(* Logix 5000 project; controller Sucrose_Main Emulate 5570 rev 20.12; software revision 20.01; part 7 of 30 *)
(* tags used below, declared in another part *)
   Alarm_ACK_Master_Timer : TIMER;
   DI_E23_5 : ALIAS FOR FLX_E23:5:I;   // Discrete Input EN2T_FLX 192.168.1.23
   DI_E25_3 : ALIAS FOR FLX_E25:3:I;   // Discrete Input EN2T_FLX 192.168.1.25
   DO_E24_2 : ALIAS FOR FLX_E24:2:O;   // Discrete Output EN2T_FLX 192.168.1.24
   DO_E25_4 : ALIAS FOR FLX_E25:4:O;   // Discrete Output EN2T_FLX 192.168.1.25
   DO_E25_5 : ALIAS FOR FLX_E25:5:O;   // Discrete Output EN2T_FLX 192.168.1.25
   FV610010_AOI : QSI_Flow_Valve;   // CIP SUPPLY TO RECEIVING PUMP #1
   FV610020_AOI : QSI_Flow_Valve;   // CIP SUPPLY TO RECEIVING PUMP #2
   FV610030_AOI : QSI_Flow_Valve;   // LOW POINT DRAIN VALVE
   FV610401_AOI : QSI_Flow_Valve;   // FV-61-04-01-O VALVE MANIFOLD TO SUCROSE TRANSFER PUMP #1 VALVE OPEN
   FV610402_AOI : QSI_Flow_Valve;   // FV-61-04-02-O VALVE MANIFOLD TO SUCROSE TRANSFER PUMP #2 VALVE OPEN
   FV620010_AOI : QSI_Flow_Valve;   // FV-62-00-10-O RECEIVING PUMP #1 TO CIP RETURN MIX PROOF VALVE OPEN
   FV620020_AOI : QSI_Flow_Valve;   // FV-62-00-20-O RECEIVING PUMP #2 TO CIP RETURN MIX PROOF VALVE OPEN
   FV620701_AOI : QSI_Flow_Valve;   // FV-62-07-01-O SUCROSE RING MAIN RETURN TO CIP RETURN VALVE VALVE OPEN
   FV621001_AOI : QSI_Flow_Valve;   // FV-62-10-01-O SUCROSE RECEIVING TO CIP RETURN VALVE OPEN
   Sucrose_MM_Enable : BOOL;
   SucroseCIP_P230401_REMOTE : CIP_REMOTE;
   SucroseCIP_P230402_REMOTE : CIP_REMOTE;
   SucroseCIP_RECEIVING2_REMOTE : CIP_REMOTE;
   SucroseCIP_RECEIVING_LINE_REMOTE : CIP_REMOTE;
   SucroseCIP_RECEIVING_REMOTE : CIP_REMOTE;
   SucroseCIP_RINGMAIN_REMOTE : CIP_REMOTE;
(* CIP_RemoteArea_EN2T_IO_Discrete_DO_E24_1, continued *)

ROUTINE MainRoutine   (* ladder *)
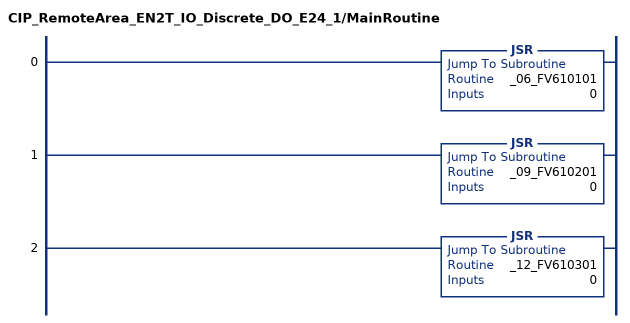
   0: JSR(_06_FV610101,0);
   1: JSR(_09_FV610201,0);
   2: JSR(_12_FV610301,0);
END_ROUTINE
END_PROGRAM

PROGRAM CIP_RemoteArea_EN2T_IO_Discrete_DO_E24_2   (* main routine MainRoutine *)

ROUTINE _00_FV610401   (* ladder *)
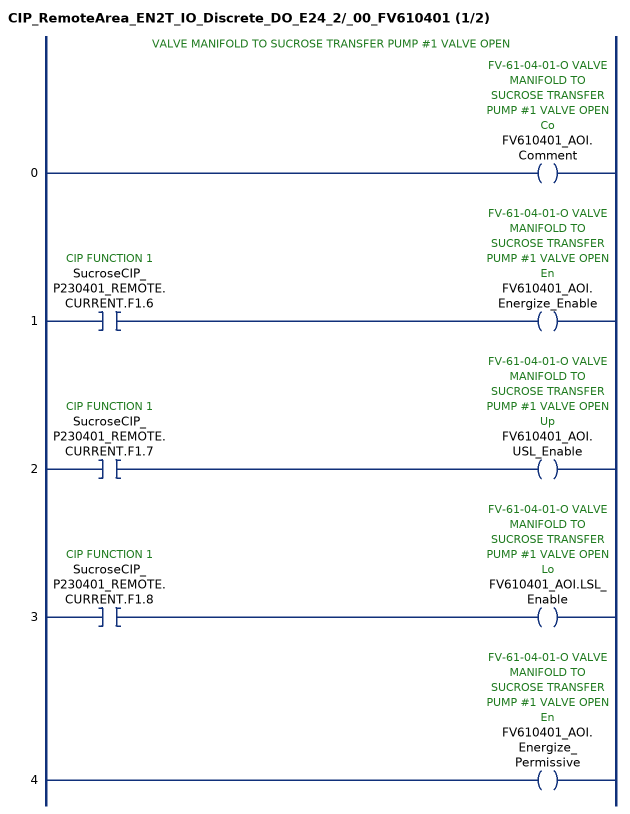
   // VALVE MANIFOLD TO SUCROSE TRANSFER PUMP #1 VALVE OPEN
   0: OTE(FV610401_AOI.Comment);
   1: XIC(SucroseCIP_P230401_REMOTE.CURRENT.F1.6)OTE(FV610401_AOI.Energize_Enable);
   2: XIC(SucroseCIP_P230401_REMOTE.CURRENT.F1.7)OTE(FV610401_AOI.USL_Enable);
   3: XIC(SucroseCIP_P230401_REMOTE.CURRENT.F1.8)OTE(FV610401_AOI.LSL_Enable);
   4: OTE(FV610401_AOI.Energize_Permissive);
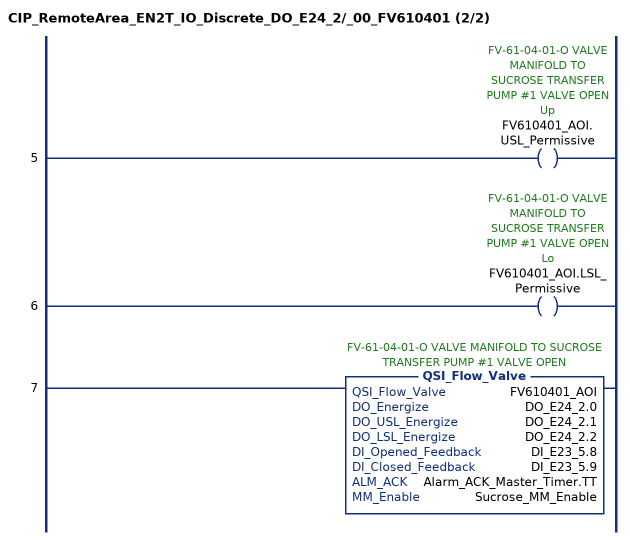
   5: OTE(FV610401_AOI.USL_Permissive);
   6: OTE(FV610401_AOI.LSL_Permissive);
   7: QSI_Flow_Valve(FV610401_AOI,DO_E24_2.0,DO_E24_2.1,DO_E24_2.2,DI_E23_5.8,DI_E23_5.9,Alarm_ACK_Master_Timer.TT,Sucrose_MM_Enable);
END_ROUTINE

ROUTINE _03_FV610402   (* ladder *)
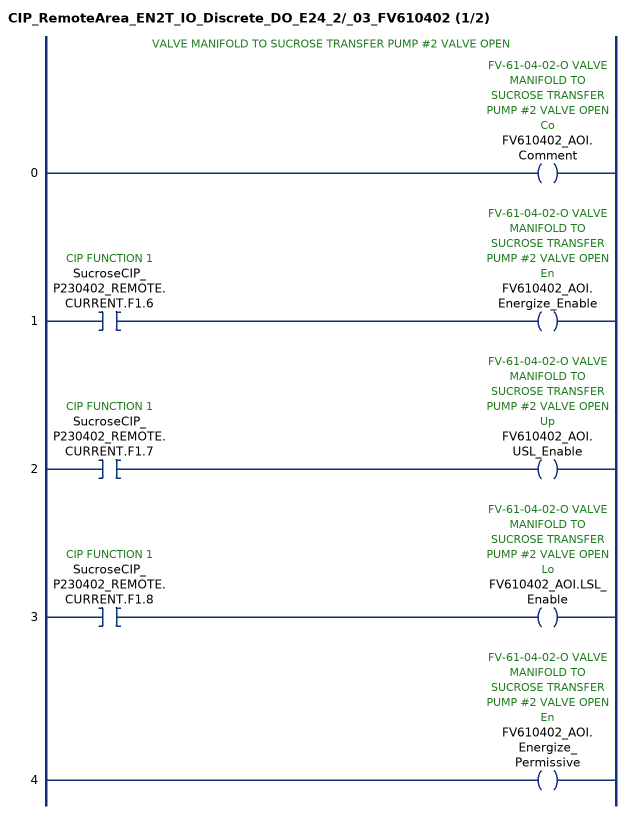
   // VALVE MANIFOLD TO SUCROSE TRANSFER PUMP #2 VALVE OPEN
   0: OTE(FV610402_AOI.Comment);
   1: XIC(SucroseCIP_P230402_REMOTE.CURRENT.F1.6)OTE(FV610402_AOI.Energize_Enable);
   2: XIC(SucroseCIP_P230402_REMOTE.CURRENT.F1.7)OTE(FV610402_AOI.USL_Enable);
   3: XIC(SucroseCIP_P230402_REMOTE.CURRENT.F1.8)OTE(FV610402_AOI.LSL_Enable);
   4: OTE(FV610402_AOI.Energize_Permissive);
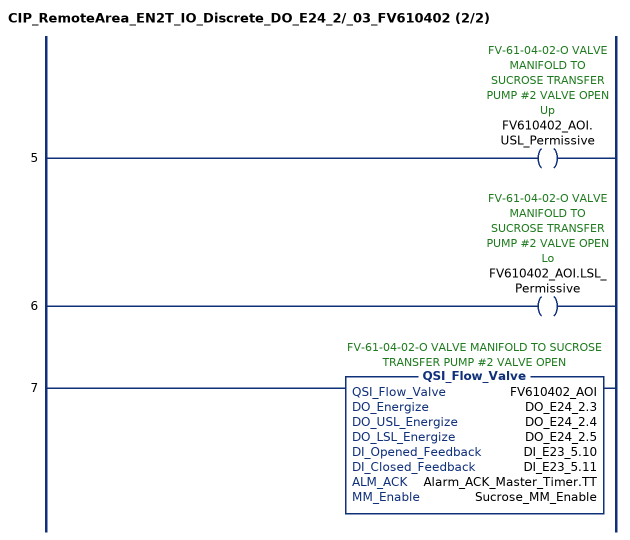
   5: OTE(FV610402_AOI.USL_Permissive);
   6: OTE(FV610402_AOI.LSL_Permissive);
   7: QSI_Flow_Valve(FV610402_AOI,DO_E24_2.3,DO_E24_2.4,DO_E24_2.5,DI_E23_5.10,DI_E23_5.11,Alarm_ACK_Master_Timer.TT,Sucrose_MM_Enable);
END_ROUTINE

ROUTINE _06_FV621001   (* ladder *)
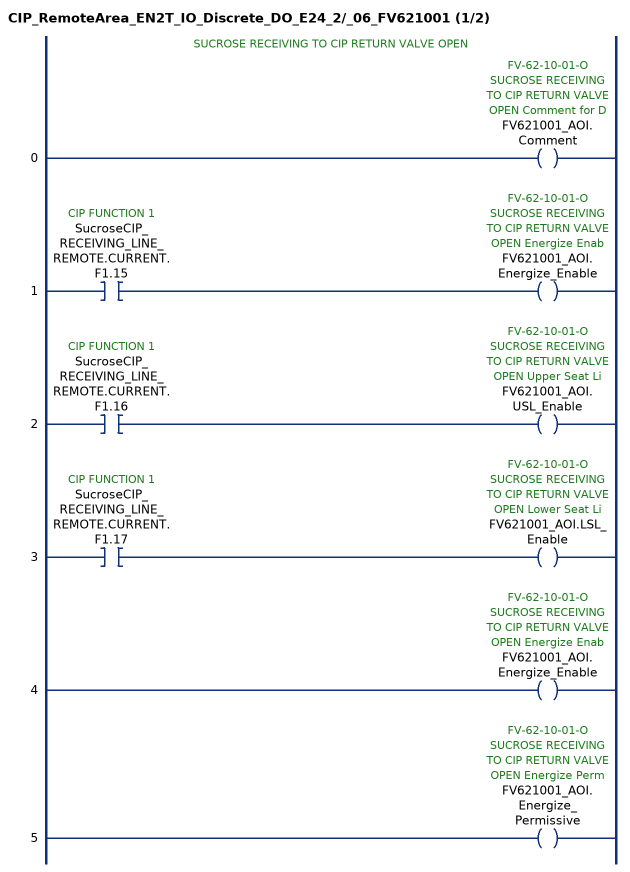
   // SUCROSE RECEIVING TO CIP RETURN VALVE OPEN
   0: OTE(FV621001_AOI.Comment);
   1: XIC(SucroseCIP_RECEIVING_LINE_REMOTE.CURRENT.F1.15)OTE(FV621001_AOI.Energize_Enable);
   2: XIC(SucroseCIP_RECEIVING_LINE_REMOTE.CURRENT.F1.16)OTE(FV621001_AOI.USL_Enable);
   3: XIC(SucroseCIP_RECEIVING_LINE_REMOTE.CURRENT.F1.17)OTE(FV621001_AOI.LSL_Enable);
   4: OTE(FV621001_AOI.Energize_Enable);
   5: OTE(FV621001_AOI.Energize_Permissive);
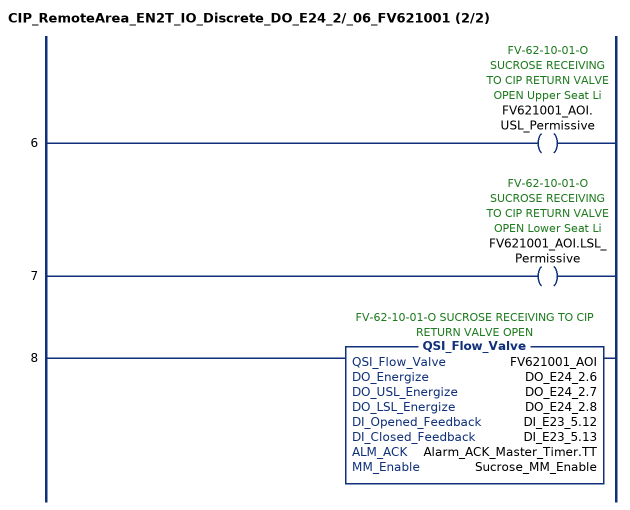
   6: OTE(FV621001_AOI.USL_Permissive);
   7: OTE(FV621001_AOI.LSL_Permissive);
   8: QSI_Flow_Valve(FV621001_AOI,DO_E24_2.6,DO_E24_2.7,DO_E24_2.8,DI_E23_5.12,DI_E23_5.13,Alarm_ACK_Master_Timer.TT,Sucrose_MM_Enable);
END_ROUTINE

ROUTINE _09_FV620701   (* ladder *)
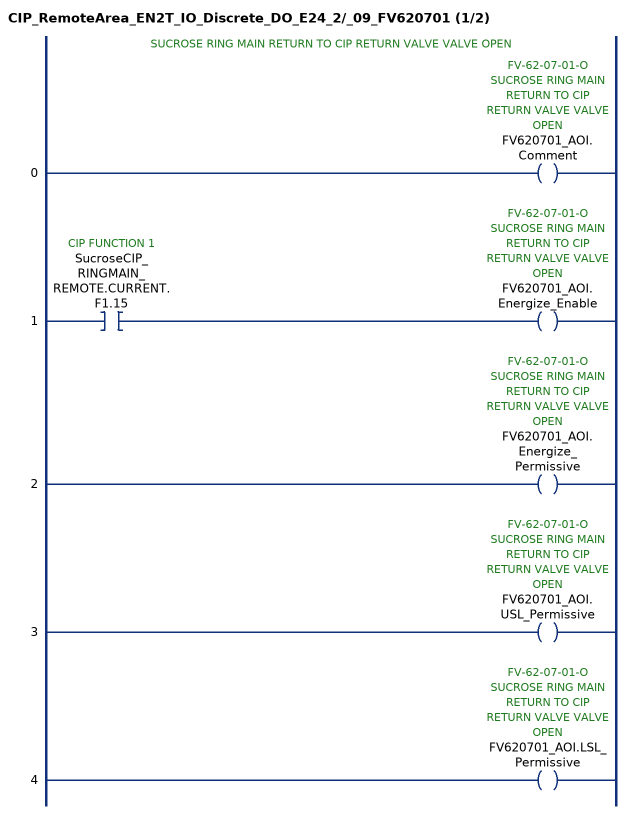
   // SUCROSE RING MAIN RETURN TO CIP RETURN VALVE VALVE OPEN
   0: OTE(FV620701_AOI.Comment);
   1: XIC(SucroseCIP_RINGMAIN_REMOTE.CURRENT.F1.15)OTE(FV620701_AOI.Energize_Enable);
   2: OTE(FV620701_AOI.Energize_Permissive);
   3: OTE(FV620701_AOI.USL_Permissive);
   4: OTE(FV620701_AOI.LSL_Permissive);
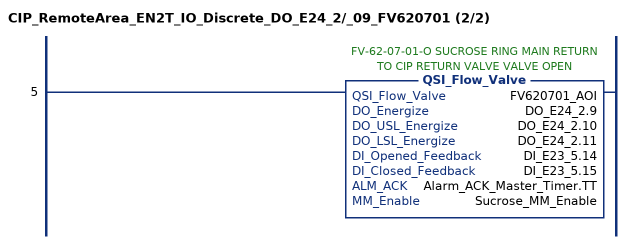
   5: QSI_Flow_Valve(FV620701_AOI,DO_E24_2.9,DO_E24_2.10,DO_E24_2.11,DI_E23_5.14,DI_E23_5.15,Alarm_ACK_Master_Timer.TT,Sucrose_MM_Enable);
END_ROUTINE

ROUTINE MainRoutine   (* ladder *)
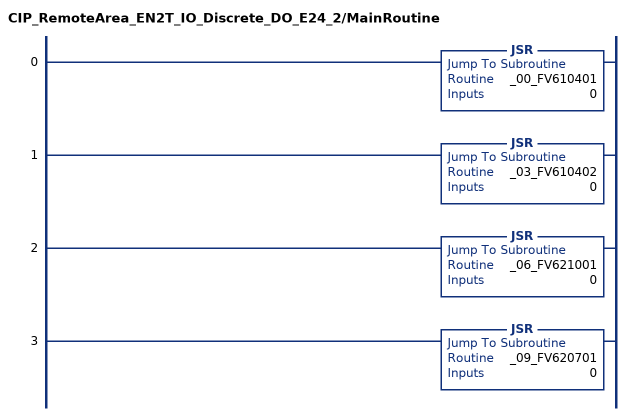
   0: JSR(_00_FV610401,0);
   1: JSR(_03_FV610402,0);
   2: JSR(_06_FV621001,0);
   3: JSR(_09_FV620701,0);
END_ROUTINE
END_PROGRAM

PROGRAM CIP_RemoteArea_EN2T_IO_Discrete_DO_E25_4   (* main routine MainRoutine *)

ROUTINE _12_FV610010   (* ladder *)
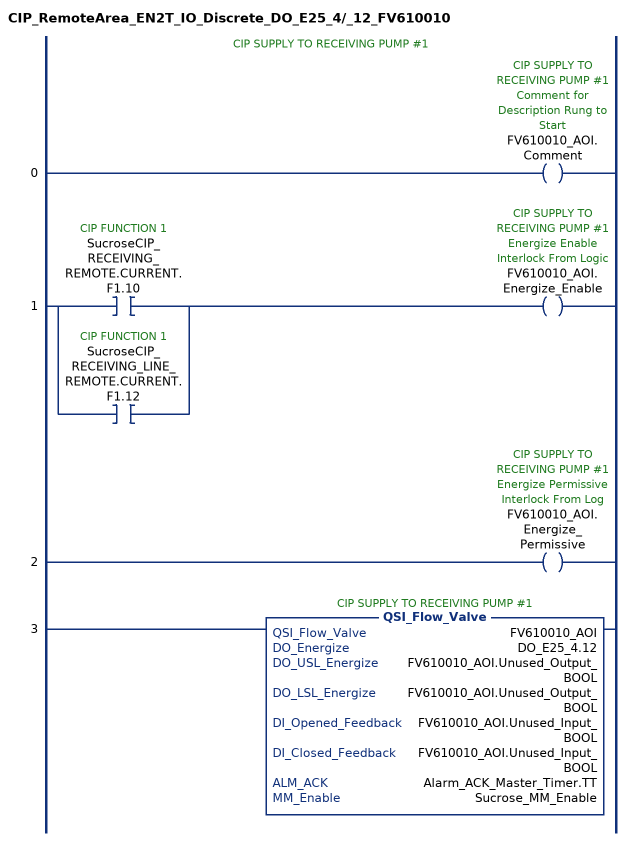
   // CIP SUPPLY TO RECEIVING PUMP #1
   0: OTE(FV610010_AOI.Comment);
   1: [XIC(SucroseCIP_RECEIVING_REMOTE.CURRENT.F1.10) ,XIC(SucroseCIP_RECEIVING_LINE_REMOTE.CURRENT.F1.12) ]OTE(FV610010_AOI.Energize_Enable);
   2: OTE(FV610010_AOI.Energize_Permissive);
   3: QSI_Flow_Valve(FV610010_AOI,DO_E25_4.12,FV610010_AOI.Unused_Output_BOOL,FV610010_AOI.Unused_Output_BOOL,FV610010_AOI.Unused_Input_BOOL,FV610010_AOI.Unused_Input_BOOL,Alarm_ACK_Master_Timer.TT,Sucrose_MM_Enable);
END_ROUTINE

ROUTINE _13_FV610020   (* ladder *)
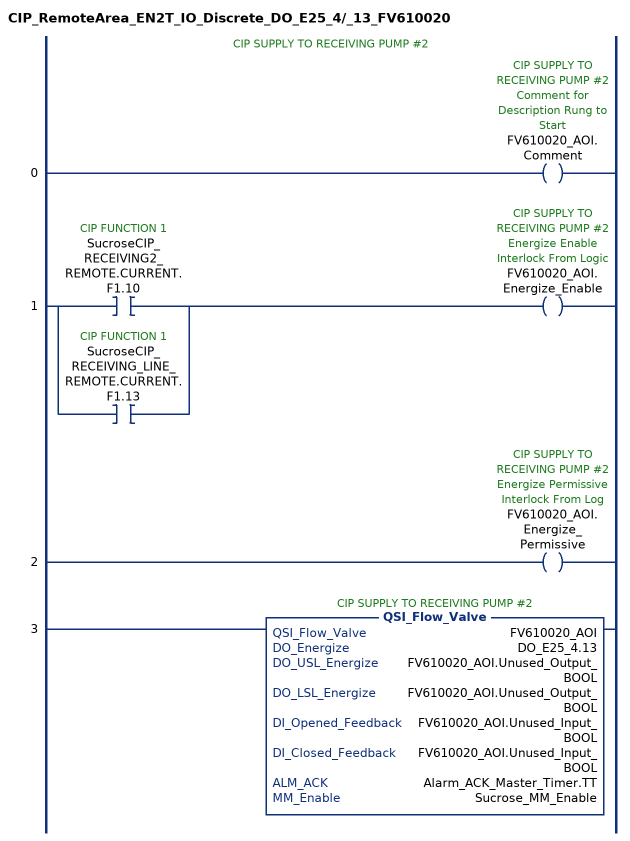
   // CIP SUPPLY TO RECEIVING PUMP #2
   0: OTE(FV610020_AOI.Comment);
   1: [XIC(SucroseCIP_RECEIVING2_REMOTE.CURRENT.F1.10) ,XIC(SucroseCIP_RECEIVING_LINE_REMOTE.CURRENT.F1.13) ]OTE(FV610020_AOI.Energize_Enable);
   2: OTE(FV610020_AOI.Energize_Permissive);
   3: QSI_Flow_Valve(FV610020_AOI,DO_E25_4.13,FV610020_AOI.Unused_Output_BOOL,FV610020_AOI.Unused_Output_BOOL,FV610020_AOI.Unused_Input_BOOL,FV610020_AOI.Unused_Input_BOOL,Alarm_ACK_Master_Timer.TT,Sucrose_MM_Enable);
END_ROUTINE

ROUTINE _14_FV610030   (* ladder *)
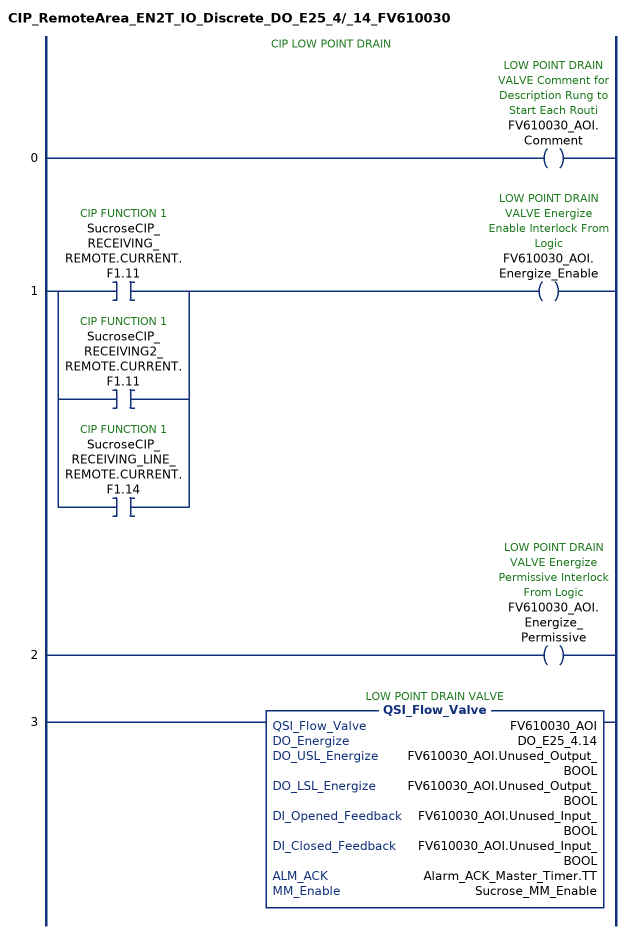
   // CIP LOW POINT DRAIN
   0: OTE(FV610030_AOI.Comment);
   1: [XIC(SucroseCIP_RECEIVING_REMOTE.CURRENT.F1.11) ,XIC(SucroseCIP_RECEIVING2_REMOTE.CURRENT.F1.11) ,XIC(SucroseCIP_RECEIVING_LINE_REMOTE.CURRENT.F1.14) ]OTE(FV610030_AOI.Energize_Enable);
   2: OTE(FV610030_AOI.Energize_Permissive);
   3: QSI_Flow_Valve(FV610030_AOI,DO_E25_4.14,FV610030_AOI.Unused_Output_BOOL,FV610030_AOI.Unused_Output_BOOL,FV610030_AOI.Unused_Input_BOOL,FV610030_AOI.Unused_Input_BOOL,Alarm_ACK_Master_Timer.TT,Sucrose_MM_Enable);
END_ROUTINE

ROUTINE MainRoutine   (* ladder *)
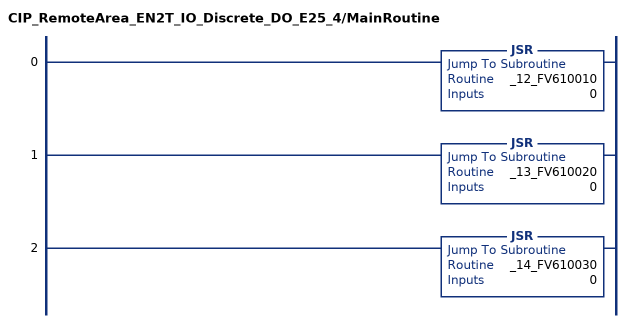
   0: JSR(_12_FV610010,0);
   1: JSR(_13_FV610020,0);
   2: JSR(_14_FV610030,0);
END_ROUTINE
END_PROGRAM

PROGRAM CIP_RemoteArea_EN2T_IO_Discrete_DO_E25_5   (* main routine MainRoutine *)

ROUTINE _06_FV620010   (* ladder *)
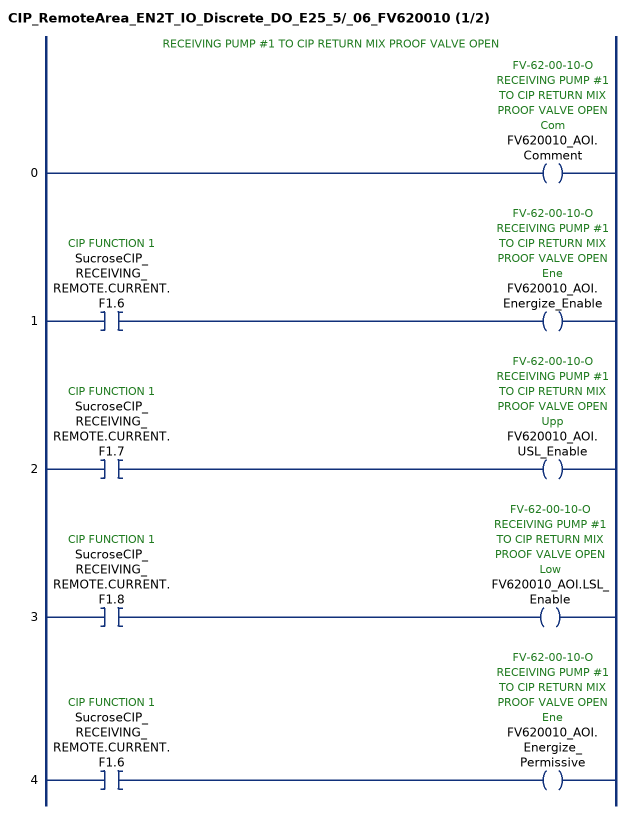
   // RECEIVING PUMP #1 TO CIP RETURN MIX PROOF VALVE OPEN
   0: OTE(FV620010_AOI.Comment);
   1: XIC(SucroseCIP_RECEIVING_REMOTE.CURRENT.F1.6)OTE(FV620010_AOI.Energize_Enable);
   2: XIC(SucroseCIP_RECEIVING_REMOTE.CURRENT.F1.7)OTE(FV620010_AOI.USL_Enable);
   3: XIC(SucroseCIP_RECEIVING_REMOTE.CURRENT.F1.8)OTE(FV620010_AOI.LSL_Enable);
   4: XIC(SucroseCIP_RECEIVING_REMOTE.CURRENT.F1.6)OTE(FV620010_AOI.Energize_Permissive);
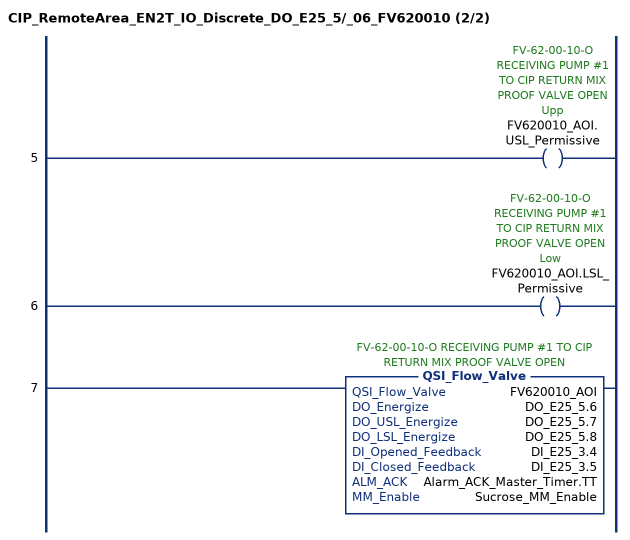
   5: OTE(FV620010_AOI.USL_Permissive);
   6: OTE(FV620010_AOI.LSL_Permissive);
   7: QSI_Flow_Valve(FV620010_AOI,DO_E25_5.6,DO_E25_5.7,DO_E25_5.8,DI_E25_3.4,DI_E25_3.5,Alarm_ACK_Master_Timer.TT,Sucrose_MM_Enable);
END_ROUTINE

ROUTINE _09_FV620020   (* ladder *)
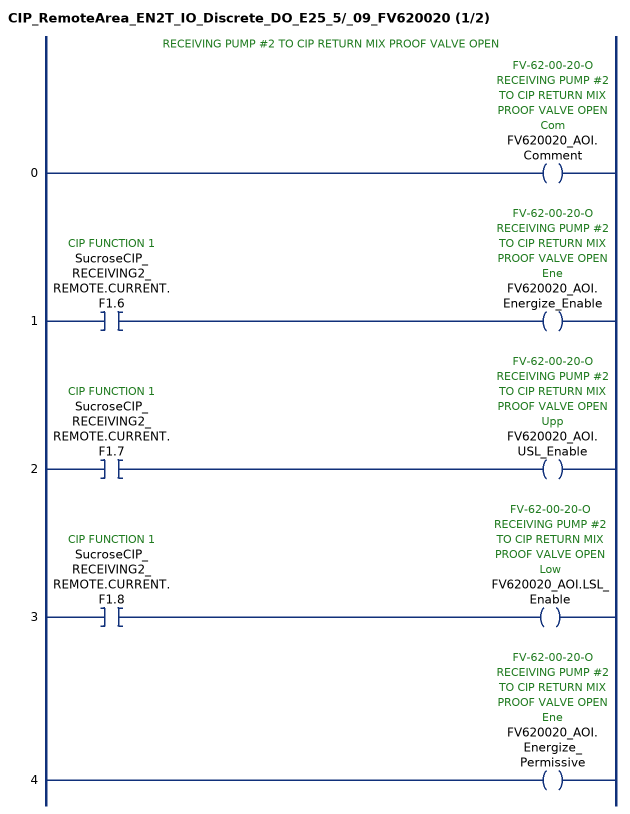
   // RECEIVING PUMP #2 TO CIP RETURN MIX PROOF VALVE OPEN
   0: OTE(FV620020_AOI.Comment);
   1: XIC(SucroseCIP_RECEIVING2_REMOTE.CURRENT.F1.6)OTE(FV620020_AOI.Energize_Enable);
   2: XIC(SucroseCIP_RECEIVING2_REMOTE.CURRENT.F1.7)OTE(FV620020_AOI.USL_Enable);
   3: XIC(SucroseCIP_RECEIVING2_REMOTE.CURRENT.F1.8)OTE(FV620020_AOI.LSL_Enable);
   4: OTE(FV620020_AOI.Energize_Permissive);
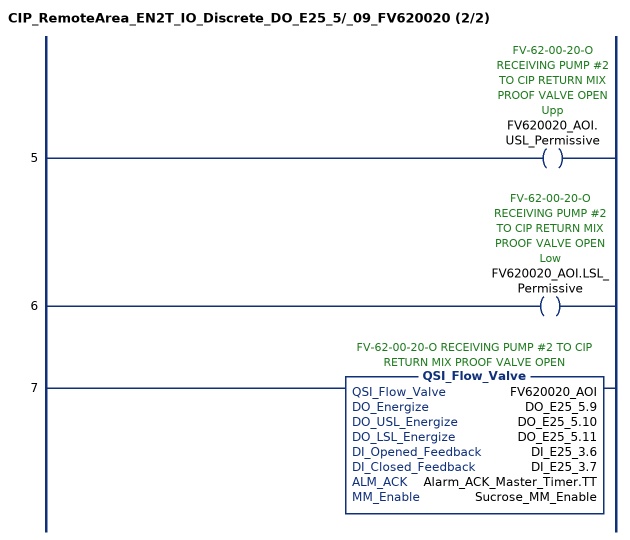
   5: OTE(FV620020_AOI.USL_Permissive);
   6: OTE(FV620020_AOI.LSL_Permissive);
   7: QSI_Flow_Valve(FV620020_AOI,DO_E25_5.9,DO_E25_5.10,DO_E25_5.11,DI_E25_3.6,DI_E25_3.7,Alarm_ACK_Master_Timer.TT,Sucrose_MM_Enable);
END_ROUTINE
